Fanuc KAREL source: kb00197.KL

-- PROVISIONAL review KL for V770-1; original PC SHA256 779bb8f7f0991329accb3f8896d77621c3f3c5120ee9ab5fcbbaba651ac8438b
-- Incomplete behavior may be omitted. Consult companion uncertainty JSON. Do not deploy.
PROGRAM KB00197
%NOLOCKGROUP
BEGIN
  -- UNRESOLVED_PC offsets 5-14; opcodes 3F,75
  -- UNRESOLVED_PC offsets 19-26; opcodes 9D,23
  -- UNRESOLVED_PC offsets 31-38; opcodes 9D,23
  -- UNRESOLVED_PC offsets 43-73; opcodes 27,22,22,2A,22,22,31
  -- UNRESOLVED_PC offsets 78-82; opcodes 7F
END KB00197
